Universal Robots PolyScope program: play_turn_6.urp

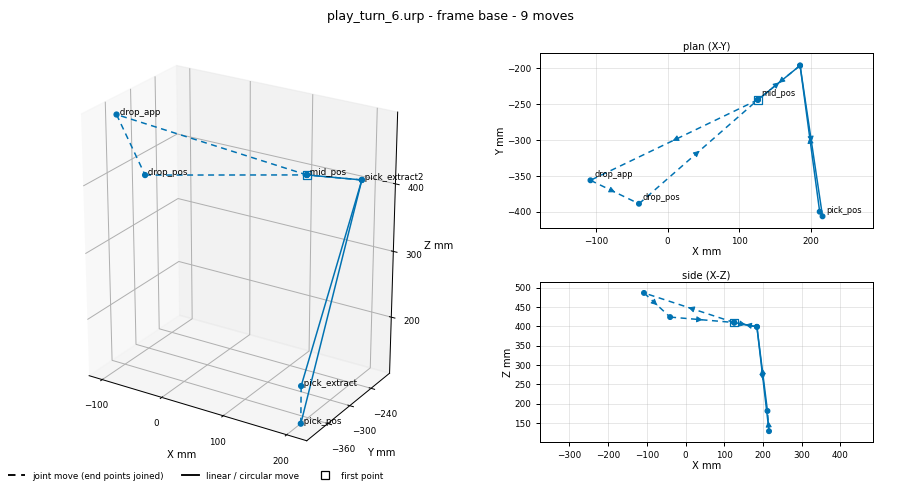
[picture p0: tool path of play_turn_6.urp in frame base, 9 of 9 moves have a stored position in this frame; points joined in program order, loops and branches not executed]
Program play_turn_6 (installation=default directory=/programs createdIn=5.5.1.82186 lastSavedIn=5.5.1.82186 robotSerialNumber=20195501773)
Calibrated DH parameters: a=[0.000078, -0.34639, -0.370501, 0.000126, 0.000068, 0]; d=[0.162438, 239.052002, -195.707731, -43.211263, 0.099699, 0.099408]; alpha=[1.569776, -0.00103, -0.002962, 1.571012, -1.570997, 0]; deltaTheta=[0, -0.617927, 6.567529, 0.333587, 0.000001, 0]
Robot Program (runOnlyOnce=false)
  URCap Gripper (Robotiq_Grippers, Robotiq Inc.) dataModel(position=0.0, force=100.0, speed=49.01960784313725, positionInDouble=0.0, forceInDouble=100.0, speedInDouble=49.01960784313725, slaveIds=[9], blocking=true)
  MoveJ speed 60 deg/s, acceleration 80 deg/s^2 (useActiveTCP=true) feature=Ref_connect4
    Waypoint mid_pos: TCP in base x=125.769 y=-243.772 z=410.19 mm, rx=2.1718 ry=2.1923 rz=-0.1426 rad; joints [89.221, -127.871, 119.758, -87.79, 268.327, 88.671] deg; TCP offset x=0 y=0 z=55 mm, rx=0 ry=0 rz=0 rad; feature pose in base x=312.569 y=-345.427 z=125.276 mm, rx=2.2161 ry=2.2035 rz=-0.0721 rad
    MoveL speed 250 mm/s, acceleration 1200 mm/s^2 (useActiveTCP=true) feature=Ref_connect4
      Waypoint pick_extract2: TCP in base x=184.495 y=-196.09 z=399.035 mm, rx=1.7798 ry=1.7673 rz=-0.5673 rad; joints [107.981, -139.662, 137.87, -128.993, 263.163, 105.834] deg; TCP offset x=0 y=0 z=55 mm, rx=0 ry=0 rz=0 rad; feature pose in base x=312.569 y=-345.427 z=125.276 mm, rx=2.2161 ry=2.2035 rz=-0.0721 rad
      Waypoint pick_pos: TCP in base x=215.75 y=-406.074 z=129.319 mm, rx=1.9558 ry=1.8112 rz=-0.5422 rad; joints [103.82, -72.219, 139.772, -190.022, 262.29, 105.838] deg
    URCap Gripper (Robotiq_Grippers, Robotiq Inc.) dataModel(position=82.74509803921569, force=100.0, speed=19.0, positionInDouble=82.74509803921569, forceInDouble=100.0, speedInDouble=19.0, slaveIds=[9], blocking=true)
    Wait Sleep waitTime=0.5
    Waypoint pick_extract: TCP in base x=211.763 y=-399.612 z=181.611 mm, rx=1.9555 ry=1.8 rz=-0.5457 rad; joints [103.474, -82.404, 139.182, -179.713, 262.4, 105.852] deg
    MoveL speed 250 mm/s, acceleration 1200 mm/s^2 (useActiveTCP=true) feature=Ref_connect4
      Waypoint pick_extract2: TCP in base x=184.495 y=-196.09 z=399.035 mm, rx=1.7798 ry=1.7673 rz=-0.5673 rad; joints [107.981, -139.662, 137.87, -128.993, 263.163, 105.834] deg
    Waypoint mid_pos: TCP in base x=125.769 y=-243.772 z=410.19 mm, rx=2.1718 ry=2.1923 rz=-0.1426 rad; joints [89.221, -127.871, 119.758, -87.79, 268.327, 88.671] deg; TCP offset x=0 y=0 z=55 mm, rx=0 ry=0 rz=0 rad; feature pose in base x=312.569 y=-345.427 z=125.276 mm, rx=2.2161 ry=2.2035 rz=-0.0721 rad
    Waypoint drop_app: TCP in base x=-107.346 y=-355.882 z=486.609 mm, rx=3.1199 ry=-0.0043 rz=0.0676 rad; joints [51.008, -108.939, 97.576, -78.027, 272.532, 141.261] deg; TCP offset x=0 y=0 z=55 mm, rx=0 ry=0 rz=0 rad
    Waypoint drop_pos: TCP in base x=-39.834 y=-388.547 z=424.233 mm, rx=3.1064 ry=0.0199 rz=0.0409 rad; joints [63.254, -107.731, 106.404, -89.777, 272.08, 152.622] deg; feature pose in base x=312.569 y=-345.427 z=125.276 mm, rx=2.2161 ry=2.2035 rz=-0.0721 rad
    URCap Gripper (Robotiq_Grippers, Robotiq Inc.) dataModel(position=70.98039215686275, force=100.0, speed=19.0, positionInDouble=70.98039215686275, forceInDouble=100.0, speedInDouble=19.0, slaveIds=[9], blocking=true)
    Wait Sleep waitTime=0.5
    URCap Gripper (Robotiq_Grippers, Robotiq Inc.) dataModel(position=0.0, force=100.0, speed=19.0, positionInDouble=0.0, forceInDouble=100.0, speedInDouble=19.0, slaveIds=[9], blocking=true)
    Waypoint mid_pos: TCP in base x=125.769 y=-243.772 z=410.19 mm, rx=2.1718 ry=2.1923 rz=-0.1426 rad; joints [89.221, -127.871, 119.758, -87.79, 268.327, 88.671] deg; TCP offset x=0 y=0 z=55 mm, rx=0 ry=0 rz=0 rad; feature pose in base x=312.569 y=-345.427 z=125.276 mm, rx=2.2161 ry=2.2035 rz=-0.0721 rad
